INTERFACE I_WashStrategy

METHOD GetDuration : TIME
VAR_INPUT
END_VAR
END_METHOD

METHOD GetProgramName : STRING
VAR_INPUT
END_VAR
END_METHOD

METHOD GetSettings : ST_WashSettings
VAR_INPUT
END_VAR
END_METHOD

METHOD Start : BOOL
VAR_INPUT
END_VAR
END_METHOD

END_INTERFACE

(* stored: Version 1.1.0.1, ProductVersion 3.1.4024.16
   Itf I_WashStrategy: Id {005279ee-3168-463d-b106-1f662ee7999c}
   Method GetDuration: Id {cb71f3c1-54db-430c-b2e1-b43e72697955}
   Method GetProgramName: Id {4e6cb005-ef5f-47ea-981d-d2a30a38056a}
   Method GetSettings: Id {f07b2014-9c96-47dc-af8e-3abf0f545366}
   Method Start: Id {0be34e3a-960f-46e0-98b5-268f5abfc757} *)
